INTERFACE I_AC

PROPERTY AC_IPAddr : STRING
GET
END_GET
END_PROPERTY

PROPERTY ACcontrol : ST_ACcontrol
GET
END_GET
END_PROPERTY

PROPERTY ACstatus : ST_ACStatus
SET
END_SET
END_PROPERTY

END_INTERFACE

(* stored: Version 1.1.0.1, ProductVersion 3.1.4024.12
   Itf I_AC: Id {cc060126-c6b2-433b-814d-4f8776017342}
   Property AC_IPAddr: Id {cfd8c9f4-33a5-4fb1-b98c-acce511c52fe}
   Get Get: Id {880535e4-b28b-4f64-b9e4-387379a70623}
   Property ACcontrol: Id {16a9f649-4679-4a86-9ab7-9ffe51e572ad}
   Get Get: Id {11c8a96d-2dcd-4202-bb7f-9fcf12f74ace}
   Property ACstatus: Id {4b9b7d4c-8109-4f9c-b4fb-d0d537c708f8}
   Set Set: Id {83cc7277-db43-4dcb-9940-a7a687579ff0} *)
